Fanuc KAREL source: kt00023.KL

-- PROVISIONAL review KL for V940-1; original PC SHA256 a2d4625943fa9fdecd64114071fbf51581c0e039830a783b7531d2558f120cb9
-- Incomplete behavior may be omitted. Consult companion uncertainty JSON. Do not deploy.
PROGRAM KT00023
%NOLOCKGROUP
VAR
  OUT : INTEGER
-- UNRESOLVED_DECL Y1 type=002018
-- UNRESOLVED_DECL H2 type=002017
BEGIN
  -- V9_ZERO_TABLE_METADATA_HINT layout=0001; no indexed target words; source/name/runtime held
  -- UNRESOLVED_PC offsets 5-19; opcodes 2E,22,9D,33,B2
  -- UNRESOLVED_PC offsets 24-38; opcodes 2E,22,9D,33,B4
  -- UNRESOLVED_PC offsets 43-68; opcodes 22,9D,33,B1,22,9D,33,B3,52,23
  -- UNRESOLVED_PC offsets 73-77; opcodes 7F
END KT00023
